FUNCTION_BLOCK FB_ShutterSafety
VAR_INPUT

    {attribute 'pytmc' := '
        pv: LSSPermission
        io: i
        field: ZNAM FALSE
        field: ONAM TRUE
    '}
    bLSSPermission : BOOL;

    {attribute 'pytmc' := '
        pv: Acknowledge
        io: io
        field: ZNAM FALSE
        field: ONAM TRUE
    '}
    bAcknowledge : BOOL;

    {attribute 'pytmc' := '
        pv: UserOpen
        io: io
        field: ZNAM Close
        field: ONAM Open
    '}
    bUserOpenRequest : BOOL;

    {attribute 'pytmc' := '
        pv: Override
        io: io
        field: ZNAM Normal mode
        field: ONAM Override mode
    '}
    bOverride : BOOL;

    nSourceIndex : UINT;
	Shutter_Enable : BOOL; 

END_VAR
VAR_IN_OUT

    (* VAR_IN_OUT -> reference to fbDestinations *)
    fbDestinations : ARRAY [1..GVL_BTPS_Constants.nDestinations] OF FB_DestinationDataStore;

END_VAR
VAR_OUTPUT

    {attribute 'pytmc' := '
        pv: Safe
        io: input
        field: ZNAM Unsafe
        field: ONAM Safe
    '}
    bSafeToOpen : BOOL;

    {attribute 'pytmc' := '
        pv: Error
        io: input
        field: ZNAM No error
        field: ONAM Error
        field: ZSV NO_ALARM
        field: OSV MAJOR
    '}
    bLatchedError : BOOL;

    {attribute 'pytmc' := '
        pv: LSS:OpenRequest
        io: input
        field: ZNAM Request close
        field: ONAM Request open
    '}
    bOpenSignal : BOOL;

    {attribute 'pytmc' := '
        pv: CurrentLD
        io: input
        field: DESC Current laser destination (LD)
        field: LOW 0
        field: HIGH 15
        field: LSV MAJOR
        field: HSV MAJOR
    '}
    nCurrentLD : INT;

    (* Rising trigger indicator of a new error condition. *)
    rtError : R_TRIG;
    (* Rising trigger indicator of user requesting override. *)
    rtOverrideSet : R_TRIG;
    (* Falling trigger for a 'close shutter' request. *)
    ftCloseRequest : F_TRIG;

END_VAR
VAR

    nDestIndex : UINT;
    bBtpsPermission : BOOL;

END_VAR


bLatchedError R= bAcknowledge;
bAcknowledge := FALSE;

// Figure out the current destination below
nCurrentLD := 0;

IF nSourceIndex >= 1 AND nSourceIndex <= GVL_BTPS_Constants.nSources THEN
    bBtpsPermission := FALSE;
    FOR nDestIndex := 1 TO GVL_BTPS_Constants.nDestinations DO
        bBtpsPermission := (
            bBtpsPermission OR
            fbDestinations[nDestIndex].stSourceDataStore[nSourceIndex].bChecksOK
        );
        IF fbDestinations[nDestIndex].stSourceDataStore[nSourceIndex].bInPosition THEN
            IF nCurrentLD = 0 THEN
                (* First "valid" destination we've seen *)
                nCurrentLD := UINT_TO_INT(nDestIndex);
            ELSE
                (* Multiple "valid" destinations? This means none are valid *)
                nCurrentLD := -1;
            END_IF
        END_IF
    END_FOR
ELSE
    bBtpsPermission := FALSE;
    bLatchedError := TRUE;
END_IF

(* Latch an error if we have no permission. *)
bLatchedError S= NOT bBtpsPermission;
rtError(CLK:=bLatchedError);

(* Reset the user open request on a new error (if not in override mode) *)
bUserOpenRequest R= rtError.Q AND NOT bOverride;

(* If the user requesets a shutter close, clear override mode. *)
ftCloseRequest(CLK:=bUserOpenRequest);
bOverride R= ftCloseRequest.Q;

(* Don't open immediately when in override mode.  Make the user request it. *)
rtOverrideSet(CLK:=bOverride);
bUserOpenRequest R= rtOverrideSet.Q AND NOT bBtpsPermission;

(* LSS permission goes low -> stop override and reset user open

NOTE: We do not have these connected yet, so we can't test this.
TODO: connect bLssPermission
TODO: Double-check logic
    bOverride R= NOT bLssPermission;
    bUserOpenRequest R= NOT bLssPermission;
*)

(* Lose permission on a latched error. *)
bBtpsPermission R= bLatchedError;

(* It's safe to open IF in override mode (user says so!) or we determined it. *)
bSafeToOpen := bOverride OR bBtpsPermission;

(* Only open the shutter if requested and it's safe. *)
bOpenSignal := bSafeToOpen AND bUserOpenRequest;

END_FUNCTION_BLOCK

(* stored: Version 1.1.0.1, ProductVersion 3.1.4022.18
   POU FB_ShutterSafety: Id {e2b40c9f-7bf0-413f-bb80-488b62056001}, SpecialFunc None *)
